// Mitsubishi GX Works2 project: LRI - PLC - SELO   PLC: Q03UDV

PROGRAM MAIN
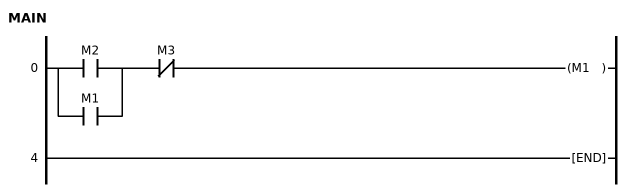
0     LD      M2
      OR      M1
      ANI     M3
      OUT     M1
4     END
END_PROGRAM
